// Mitsubishi GX Works2 project: data resister with timer   PLC: FX1N/FX1NC

PROGRAM MAIN
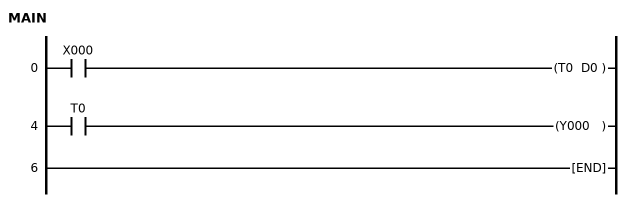
0     LD      X000
      OUT     T0 D0
4     LD      T0
      OUT     Y000
6     END
END_PROGRAM
